PROGRAM MAIN
VAR
		fbWatershed: Watershed();

END_VAR

fbWatershed();

END_PROGRAM

(* stored: Version 1.1.0.1, ProductVersion 3.1.4024.12
   POU MAIN: Id {d34730a9-7962-4660-a315-ab178b033e97}, SpecialFunc None *)
